// TIA Portal V18 export
DATA_BLOCK "Control_Buttons_Activation_DB"   // DB89
VERSION : 0.1
// stored: AutoNumber true, DBAccessibleFromOPCUA true, InstanceOfName Control_Buttons_Activation, InstanceOfType FB
"Control_Buttons_Activation"
   // VAR_INPUT
   //    JogInZ1pos : Bool;
   //    JogInZ1neg : Bool;
   //    JogInZ2pos : Bool;
   //    JogInZ2neg : Bool;
   // END_VAR
   // VAR_OUTPUT
   //    Control_Buttons_Move_Permission : Bool;
   //    Control_Buttons_ActivatedOUT : Bool;
   // END_VAR
   // VAR
   //    Step01 : Bool;
   //    Step02 : Bool;
   //    Step03 : Bool;
   //    Step04 : Bool;
   //    Step05 : Bool;
   //    Step06 : Bool;
   //    Step07 : Bool;
   //    Step08 : Bool;
   //    AnyButtonPressed : Bool;
   //    AllButtonsPressed : Bool;
   //    ControlButtonsActivated : Bool;
   // END_VAR
BEGIN
END_DATA_BLOCK
